FUNCTION_BLOCK FB_Motion


VAR_INPUT

bPowerX       : BOOL;;

bPowerY       : BOOL;;

bPowerZ       : BOOL;;

bPowerN       : BOOL;;


bStopX        : BOOL;;

bStopY        : BOOL;;

bStopZ        : BOOL;;

bStopN        : BOOL;;


bAbsX         : BOOL;;

bAbsY         : BOOL;;

bAbsZ         : BOOL;;


bVelN         : BOOL;;


bResetX       : BOOL;;

bResetY       : BOOL;;

bResetZ       : BOOL;;

bResetN       : BOOL;;


bSetPosN      : BOOL;;


bHaltN        : BOOL;;

bHaltX        : BOOL;;

bHaltY        : BOOL;;

bHaltZ        : BOOL;;


mcPowerX,;
        mcPowerY,;
        mcPowerZ,;
        mcPowerN      : MC_Power;;


mcStopX,;
        mcStopY,;
        mcStopZ,;
        mcStopN       : MC_Stop;;


mcMoveabsX,;
        mcMoveabsY,;
        mcMoveabsZ    : MC_MoveAbsolute;;


mcMoveVelN    : MC_MoveVelocity;;


mcResetX,;
        mcResetY,;
        mcResetZ,;
        mcResetN      : MC_Reset;;


mcSetPostionN : MC_SetPosition;;

mcHaltN,;
        mcHaltX,;
        mcHaltY,;
        mcHaltZ       : MC_Halt;;

    END_VAR


VAR_OUTPUT

    END_VAR


VAR





    END_VAR

END_FUNCTION_BLOCK

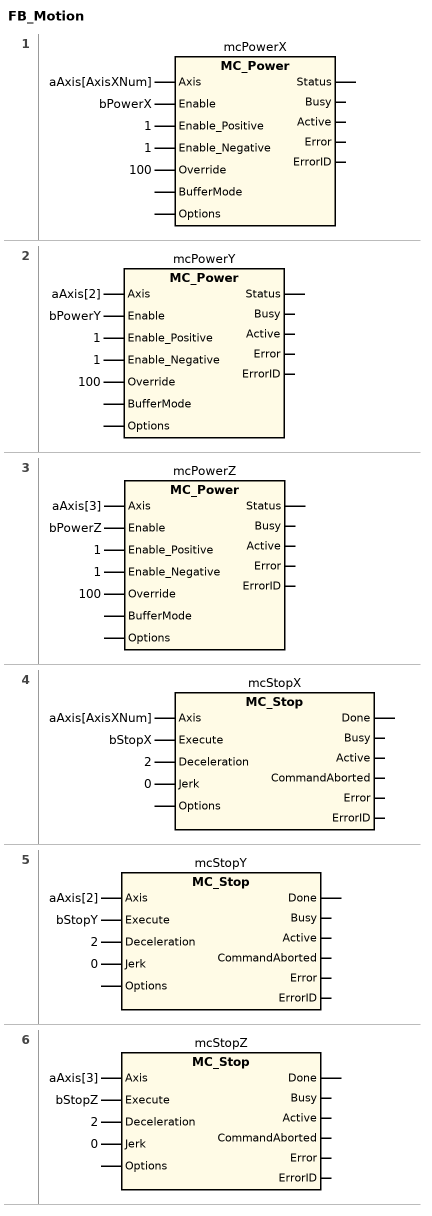
// NETWORK 1
mcPowerX(
    Axis := aAxis[AxisXNum],
    Enable := bPowerX,
    Enable_Positive := 1,
    Enable_Negative := 1,
    Override := 100); // MC_Power

// NETWORK 2
mcPowerY(Axis := aAxis[2], Enable := bPowerY, Enable_Positive := 1, Enable_Negative := 1, Override := 100); // MC_Power

// NETWORK 3
mcPowerZ(Axis := aAxis[3], Enable := bPowerZ, Enable_Positive := 1, Enable_Negative := 1, Override := 100); // MC_Power

// NETWORK 4
mcStopX(Axis := aAxis[AxisXNum], Execute := bStopX, Deceleration := 2, Jerk := 0); // MC_Stop

// NETWORK 5
mcStopY(Axis := aAxis[2], Execute := bStopY, Deceleration := 2, Jerk := 0); // MC_Stop

// NETWORK 6
mcStopZ(Axis := aAxis[3], Execute := bStopZ, Deceleration := 2, Jerk := 0); // MC_Stop

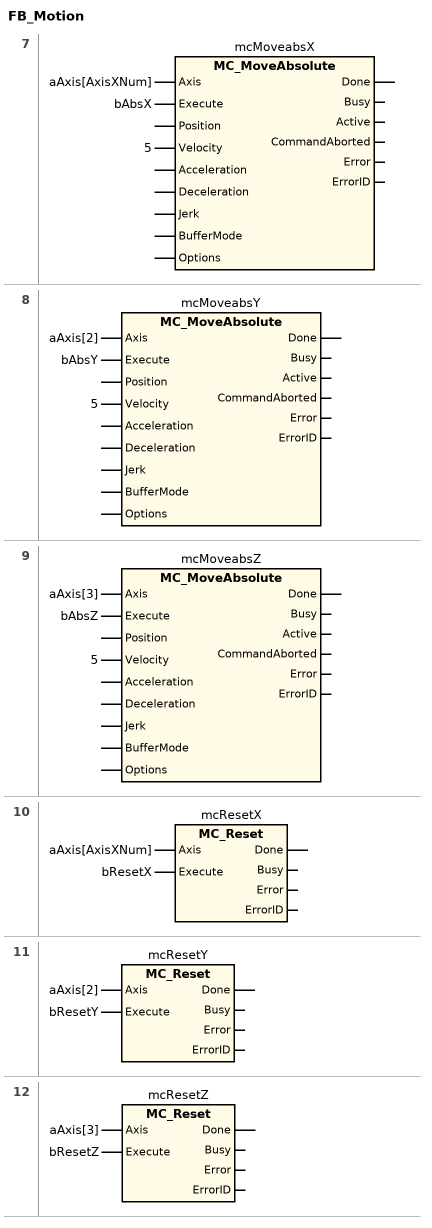
// NETWORK 7
mcMoveabsX(Axis := aAxis[AxisXNum], Execute := bAbsX, Velocity := 5); // MC_MoveAbsolute

// NETWORK 8
mcMoveabsY(Axis := aAxis[2], Execute := bAbsY, Velocity := 5); // MC_MoveAbsolute

// NETWORK 9
mcMoveabsZ(Axis := aAxis[3], Execute := bAbsZ, Velocity := 5); // MC_MoveAbsolute

// NETWORK 10
mcResetX(Axis := aAxis[AxisXNum], Execute := bResetX); // MC_Reset

// NETWORK 11
mcResetY(Axis := aAxis[2], Execute := bResetY); // MC_Reset

// NETWORK 12
mcResetZ(Axis := aAxis[3], Execute := bResetZ); // MC_Reset

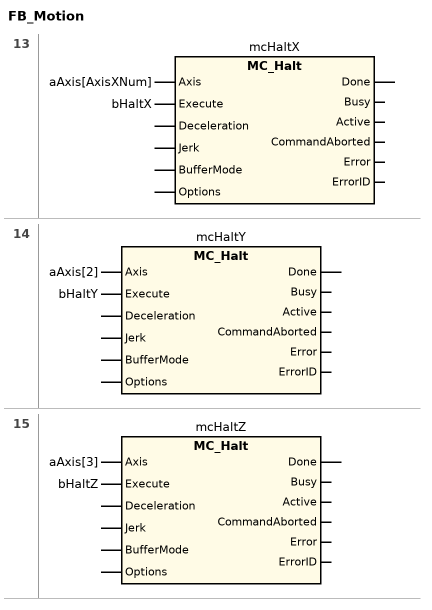
// NETWORK 13
mcHaltX(Axis := aAxis[AxisXNum], Execute := bHaltX); // MC_Halt

// NETWORK 14
mcHaltY(Axis := aAxis[2], Execute := bHaltY); // MC_Halt

// NETWORK 15
mcHaltZ(Axis := aAxis[3], Execute := bHaltZ); // MC_Halt

END_FUNCTION_BLOCK

(* stored: Version 1.1.0.1, ProductVersion 3.1.4024.12
   POU FB_Motion: Id {0e7c8735-3071-4e42-8b84-3565d03b8ea4}, SpecialFunc None *)
